// TwinCAT 3 PLC project CutomKeypadPLC
// ProgramVersion: 3.1.4023.0
// CompilerDefines: VISU_USEWSTRING
// libraries:
//   Tc2_Standard, * (Beckhoff Automation GmbH)
//   Tc2_System, * (Beckhoff Automation GmbH)
//   Tc3_Module, * (Beckhoff Automation GmbH)
//   VisuDialogs, * (System)
//   VisuSymbols,3.5.10.0,System
// project tree:
//   / GlobalTextList.TcGTLO, PlcTask.TcTTO, Visualization Manager.TcVMO (not stored), VISU_TASK.TcTTO
//   POUs/ MAIN.TcPOU
//   VISUs/ Custom_Keypad.TcVIS, Custom_Numpad.TcVIS, Visualization.TcVIS
// real-time tasks:
//   TASK PlcTask: cycle T#10ms, priority 20, ADS port 350
//   TASK VISU_TASK: cycle T#200000us, priority 30, ADS port 351

CONFIGURATION CutomKeypadPLC
    RESOURCE PLC ON TwinCAT3
        TASK PlcTask(INTERVAL := T#10ms, PRIORITY := 20);
        TASK VISU_TASK(INTERVAL := T#200000us, PRIORITY := 30);
        PROGRAM MAIN WITH PlcTask : MAIN;
        PROGRAM VisuElems_Visu_Prg WITH VISU_TASK : VisuElems.Visu_Prg;
    END_RESOURCE
END_CONFIGURATION

// ---- POUs/MAIN.TcPOU
(*	| author		| Beckhoff Automation Poland	|	*)
(* 	-------------------------------------------------	*)
(*	| wersion		| 1.0							|	*)
(* 	-------------------------------------------------	*)
(*	| TC version	| 3.1.4024.7					| 	*)
(* 	-------------------------------------------------	*)
(*	| date			| 19.05.2020					|	*)
(* 	-------------------------------------------------	*)
(*	| description	| custom keypad with hotkeys	|  	*)

PROGRAM MAIN
VAR
	iTest 	: INT;
	sTest	: STRING;
END_VAR

END_PROGRAM

// ---- GlobalTextList.TcGTLO
TEXTLIST GlobalTextList
  338 = '!'
  340 = '"'
  991 = '#'
  344 = '$'
  346 = '%'
  189 = '%s'
  169 = '&'
  992 = "'"
  174 = '('
  177 = ')'
  333 = '*'
  332 = '+'
  90 = '+/-'
  153 = ','
  157 = '-'
  155 = '.'
  171 = '/'
  179 = '0'
  337 = '1'
  339 = '2'
  341 = '3'
  343 = '4'
  345 = '5'
  347 = '6'
  170 = '7'
  172 = '8'
  176 = '9'
  156 = ':'
  154 = ';'
  137 = '<'
  181 = '='
  138 = '>'
  184 = '?'
  993 = '@'
  160 = 'a'
  161 = 'A'
  147 = 'b'
  148 = 'B'
  781 = 'Back'
  92 = 'Backspace'
  143 = 'c'
  144 = 'C'
  780 = 'Clear'
  164 = 'd'
  974 = 'D'
  998 = 'e'
  999 = 'E'
  253 = 'Enter number: %i'
  452 = 'Enter text: %s'
  779 = 'ESC'
  975 = 'f'
  976 = 'F'
  977 = 'g'
  978 = 'G'
  979 = 'h'
  980 = 'H'
  1008 = 'i'
  1009 = 'I'
  981 = 'j'
  982 = 'J'
  983 = 'k'
  984 = 'K'
  985 = 'l'
  986 = 'L'
  151 = 'm'
  152 = 'M'
  192 = 'Max:'
  191 = 'Min:'
  149 = 'n'
  150 = 'N'
  1010 = 'o'
  1011 = 'O'
  778 = 'OK'
  1012 = 'p'
  1013 = 'P'
  994 = 'q'
  995 = 'Q'
  1000 = 'r'
  1001 = 'R'
  162 = 's'
  163 = 'S'
  782 = 'Shift'
  783 = 'Space'
  1002 = 't'
  1003 = 'T'
  1006 = 'u'
  1007 = 'U'
  145 = 'v'
  146 = 'V'
  996 = 'w'
  997 = 'W'
  141 = 'x'
  142 = 'X'
  139 = 'y'
  140 = 'Y'
  1004 = 'z'
  1005 = 'Z'
  787 = '['
  187 = '\\'
  788 = ']'
  335 = '^'
  158 = '_'
  786 = '{'
  790 = '|'
  789 = '}'
  334 = '~'
  108 = '§'
  84 = '°'
  19 = '²'
  23 = '³'
  186 = '´'
  35 = 'ä'
  81 = 'Ä'
  29 = 'ö'
  34 = 'Ö'
  82 = 'ü'
  83 = 'Ü'
  109 = 'ß'
  28 = '€'
END_TEXTLIST

// ---- VISUs/Custom_Keypad.TcVIS
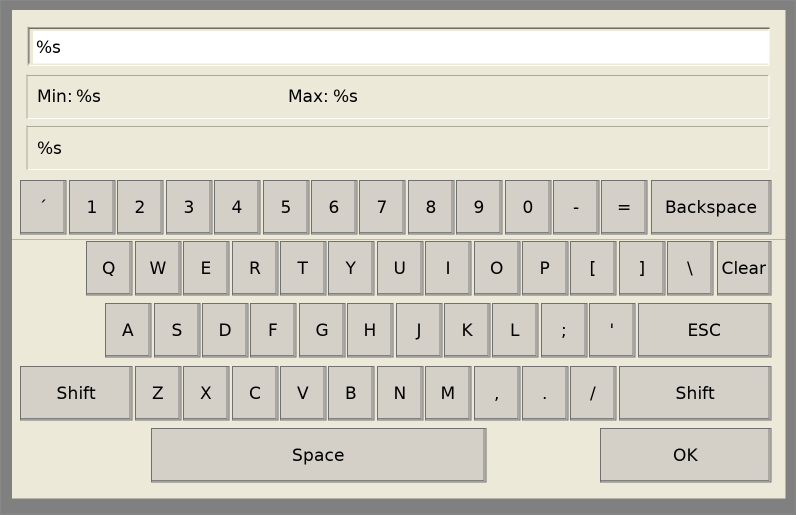
VISUALIZATION Custom_Keypad  // 796x515
VAR_INPUT
	stVariableValue : STRING;
	stMin : STRING;
	stMax : STRING;
	stTitle : STRING;
	flags : DWORD;
END_VAR
VAR
	bInit : BOOL;
	bShift : BOOL;
	stMessage : STRING;
	stOutputValue : STRING;
END_VAR
    Rectangle (0,0 796x515)
    Rectangle (12,169 773x70)
    Rectangle (12,240 773x62)
    Rectangle (12,301 773x63)
    Rectangle (12,364 773x62)
    Rectangle (12,423 773x75)
    Button (600,428 171x54), "OK"
        OnMouseDown: CloseDialog Dialog=Custom_Keypad, Result=OK, NumpadKeypad=True, NumpadKeypadSet=True
    Button (638,303 133x54), "ESC"
        OnMouseDown: CloseDialog Dialog=Custom_Keypad, Result=Cancel, NumpadKeypad=True, NumpadKeypadSet=True
    Button (717,241 54x54), "Clear"
        OnMouseDown: execute { stVariableValue := ''; stOutputValue := ''; }
    Button (651,180 120x54), "Backspace"
        OnMouseDown: execute { VisuDlg_CheckedBack(stOutputValue, stVariableValue, bInit); }
    Button (619,366 152x54), "Shift"
        OnMouseDown: toggle bShift
    Button (151,428 335x54), "Space"
        OnMouseDown: execute { VisuDlg_CheckedAppend(stOutputValue, stVariableValue, bInit, (flags AND VisuElems.Visu_InputFlags.Password) = 1, ' '); }
    Button (667,241 46x54), "|", invisible if: NOT bShift
        OnMouseDown: execute { VisuDlg_CheckedAppend(stOutputValue, stVariableValue, bInit, (flags AND VisuElems.Visu_InputFlags.Password) = 1, '|'); }
    Button (474,366 46x54), "<", invisible if: NOT bShift
        OnMouseDown: execute { VisuDlg_CheckedAppend(stOutputValue, stVariableValue, bInit, (flags AND VisuElems.Visu_InputFlags.Password) = 1, '<'); }
    Button (522,366 46x54), ">", invisible if: NOT bShift
        OnMouseDown: execute { VisuDlg_CheckedAppend(stOutputValue, stVariableValue, bInit, (flags AND VisuElems.Visu_InputFlags.Password) = 1, '>'); }
    Button (328,241 46x54), "y", invisible if: NOT bShift
        OnMouseDown: execute { VisuDlg_CheckedAppend(stOutputValue, stVariableValue, bInit, (flags AND VisuElems.Visu_InputFlags.Password) = 1, 'y'); }
    Button (328,241 46x54), "Y", invisible if: bShift
        OnMouseDown: execute { VisuDlg_CheckedAppend(stOutputValue, stVariableValue, bInit, (flags AND VisuElems.Visu_InputFlags.Password) = 1, 'Y'); }
    Button (183,366 46x54), "x", invisible if: NOT bShift
        OnMouseDown: execute { VisuDlg_CheckedAppend(stOutputValue, stVariableValue, bInit, (flags AND VisuElems.Visu_InputFlags.Password) = 1, 'x'); }
    Button (183,366 46x54), "X", invisible if: bShift
        OnMouseDown: execute { VisuDlg_CheckedAppend(stOutputValue, stVariableValue, bInit, (flags AND VisuElems.Visu_InputFlags.Password) = 1, 'X'); }
    Button (232,366 46x54), "c", invisible if: NOT bShift
        OnMouseDown: execute { VisuDlg_CheckedAppend(stOutputValue, stVariableValue, bInit, (flags AND VisuElems.Visu_InputFlags.Password) = 1, 'c'); }
    Button (232,366 46x54), "C", invisible if: bShift
        OnMouseDown: execute { VisuDlg_CheckedAppend(stOutputValue, stVariableValue, bInit, (flags AND VisuElems.Visu_InputFlags.Password) = 1, 'C'); }
    Button (280,366 46x54), "v", invisible if: NOT bShift
        OnMouseDown: execute { VisuDlg_CheckedAppend(stOutputValue, stVariableValue, bInit, (flags AND VisuElems.Visu_InputFlags.Password) = 1, 'v'); }
    Button (280,366 46x54), "V", invisible if: bShift
        OnMouseDown: execute { VisuDlg_CheckedAppend(stOutputValue, stVariableValue, bInit, (flags AND VisuElems.Visu_InputFlags.Password) = 1, 'V'); }
    Button (328,366 46x54), "b", invisible if: NOT bShift
        OnMouseDown: execute { VisuDlg_CheckedAppend(stOutputValue, stVariableValue, bInit, (flags AND VisuElems.Visu_InputFlags.Password) = 1, 'b'); }
    Button (328,366 46x54), "B", invisible if: bShift
        OnMouseDown: execute { VisuDlg_CheckedAppend(stOutputValue, stVariableValue, bInit, (flags AND VisuElems.Visu_InputFlags.Password) = 1, 'B'); }
    Button (377,366 46x54), "n", invisible if: NOT bShift
        OnMouseDown: execute { VisuDlg_CheckedAppend(stOutputValue, stVariableValue, bInit, (flags AND VisuElems.Visu_InputFlags.Password) = 1, 'n'); }
    Button (377,366 46x54), "N", invisible if: bShift
        OnMouseDown: execute { VisuDlg_CheckedAppend(stOutputValue, stVariableValue, bInit, (flags AND VisuElems.Visu_InputFlags.Password) = 1, 'N'); }
    Button (425,366 46x54), "m", invisible if: NOT bShift
        OnMouseDown: execute { VisuDlg_CheckedAppend(stOutputValue, stVariableValue, bInit, (flags AND VisuElems.Visu_InputFlags.Password) = 1, 'm'); }
    Button (425,366 46x54), "M", invisible if: bShift
        OnMouseDown: execute { VisuDlg_CheckedAppend(stOutputValue, stVariableValue, bInit, (flags AND VisuElems.Visu_InputFlags.Password) = 1, 'M'); }
    Button (541,303 46x54), ":", invisible if: NOT bShift
        OnMouseDown: execute { VisuDlg_CheckedAppend(stOutputValue, stVariableValue, bInit, (flags AND VisuElems.Visu_InputFlags.Password) = 1, ':'); }
    Button (553,180 46x54), "_", invisible if: NOT bShift
        OnMouseDown: execute { VisuDlg_CheckedAppend(stOutputValue, stVariableValue, bInit, (flags AND VisuElems.Visu_InputFlags.Password) = 1, '_'); }
    Button (105,303 46x54), "a", invisible if: NOT bShift
        OnMouseDown: execute { VisuDlg_CheckedAppend(stOutputValue, stVariableValue, bInit, (flags AND VisuElems.Visu_InputFlags.Password) = 1, 'a'); }
    Button (105,303 46x54), "A", invisible if: bShift
        OnMouseDown: execute { VisuDlg_CheckedAppend(stOutputValue, stVariableValue, bInit, (flags AND VisuElems.Visu_InputFlags.Password) = 1, 'A'); }
    Button (154,303 46x54), "s", invisible if: NOT bShift
        OnMouseDown: execute { VisuDlg_CheckedAppend(stOutputValue, stVariableValue, bInit, (flags AND VisuElems.Visu_InputFlags.Password) = 1, 's'); }
    Button (154,303 46x54), "S", invisible if: bShift
        OnMouseDown: execute { VisuDlg_CheckedAppend(stOutputValue, stVariableValue, bInit, (flags AND VisuElems.Visu_InputFlags.Password) = 1, 'S'); }
    Button (202,303 46x54), "d", invisible if: NOT bShift
        OnMouseDown: execute { VisuDlg_CheckedAppend(stOutputValue, stVariableValue, bInit, (flags AND VisuElems.Visu_InputFlags.Password) = 1, 'd'); }
    Button (202,303 46x54), "D", invisible if: bShift
        OnMouseDown: execute { VisuDlg_CheckedAppend(stOutputValue, stVariableValue, bInit, (flags AND VisuElems.Visu_InputFlags.Password) = 1, 'D'); }
    Button (250,303 46x54), "f", invisible if: NOT bShift
        OnMouseDown: execute { VisuDlg_CheckedAppend(stOutputValue, stVariableValue, bInit, (flags AND VisuElems.Visu_InputFlags.Password) = 1, 'f'); }
    Button (250,303 46x54), "F", invisible if: bShift
        OnMouseDown: execute { VisuDlg_CheckedAppend(stOutputValue, stVariableValue, bInit, (flags AND VisuElems.Visu_InputFlags.Password) = 1, 'F'); }
    Button (299,303 46x54), "g", invisible if: NOT bShift
        OnMouseDown: execute { VisuDlg_CheckedAppend(stOutputValue, stVariableValue, bInit, (flags AND VisuElems.Visu_InputFlags.Password) = 1, 'g'); }
    Button (299,303 46x54), "G", invisible if: bShift
        OnMouseDown: execute { VisuDlg_CheckedAppend(stOutputValue, stVariableValue, bInit, (flags AND VisuElems.Visu_InputFlags.Password) = 1, 'G'); }
    Button (347,303 46x54), "h", invisible if: NOT bShift
        OnMouseDown: execute { VisuDlg_CheckedAppend(stOutputValue, stVariableValue, bInit, (flags AND VisuElems.Visu_InputFlags.Password) = 1, 'h'); }
    Button (347,303 46x54), "H", invisible if: bShift
        OnMouseDown: execute { VisuDlg_CheckedAppend(stOutputValue, stVariableValue, bInit, (flags AND VisuElems.Visu_InputFlags.Password) = 1, 'H'); }
    Button (396,303 46x54), "j", invisible if: NOT bShift
        OnMouseDown: execute { VisuDlg_CheckedAppend(stOutputValue, stVariableValue, bInit, (flags AND VisuElems.Visu_InputFlags.Password) = 1, 'j'); }
    Button (396,303 46x54), "J", invisible if: bShift
        OnMouseDown: execute { VisuDlg_CheckedAppend(stOutputValue, stVariableValue, bInit, (flags AND VisuElems.Visu_InputFlags.Password) = 1, 'J'); }
    Button (444,303 46x54), "k", invisible if: NOT bShift
        OnMouseDown: execute { VisuDlg_CheckedAppend(stOutputValue, stVariableValue, bInit, (flags AND VisuElems.Visu_InputFlags.Password) = 1, 'k'); }
    Button (444,303 46x54), "K", invisible if: bShift
        OnMouseDown: execute { VisuDlg_CheckedAppend(stOutputValue, stVariableValue, bInit, (flags AND VisuElems.Visu_InputFlags.Password) = 1, 'K'); }
    Button (492,303 46x54), "l", invisible if: NOT bShift
        OnMouseDown: execute { VisuDlg_CheckedAppend(stOutputValue, stVariableValue, bInit, (flags AND VisuElems.Visu_InputFlags.Password) = 1, 'l'); }
    Button (492,303 46x54), "L", invisible if: bShift
        OnMouseDown: execute { VisuDlg_CheckedAppend(stOutputValue, stVariableValue, bInit, (flags AND VisuElems.Visu_InputFlags.Password) = 1, 'L'); }
    Button (166,180 46x54), "#", invisible if: NOT bShift
        OnMouseDown: execute { VisuDlg_CheckedAppend(stOutputValue, stVariableValue, bInit, (flags AND VisuElems.Visu_InputFlags.Password) = 1, '#'); }
    Button (117,180 46x54), "@", invisible if: NOT bShift
        OnMouseDown: execute { VisuDlg_CheckedAppend(stOutputValue, stVariableValue, bInit, (flags AND VisuElems.Visu_InputFlags.Password) = 1, '@'); }
    Button (86,241 46x54), "q", invisible if: NOT bShift
        OnMouseDown: execute { VisuDlg_CheckedAppend(stOutputValue, stVariableValue, bInit, (flags AND VisuElems.Visu_InputFlags.Password) = 1, 'q'); }
    Button (86,241 46x54), "Q", invisible if: bShift
        OnMouseDown: execute { VisuDlg_CheckedAppend(stOutputValue, stVariableValue, bInit, (flags AND VisuElems.Visu_InputFlags.Password) = 1, 'Q'); }
    Button (135,241 46x54), "w", invisible if: NOT bShift
        OnMouseDown: execute { VisuDlg_CheckedAppend(stOutputValue, stVariableValue, bInit, (flags AND VisuElems.Visu_InputFlags.Password) = 1, 'w'); }
    Button (135,241 46x54), "W", invisible if: bShift
        OnMouseDown: execute { VisuDlg_CheckedAppend(stOutputValue, stVariableValue, bInit, (flags AND VisuElems.Visu_InputFlags.Password) = 1, 'W'); }
    Button (183,241 46x54), "e", invisible if: NOT bShift
        OnMouseDown: execute { VisuDlg_CheckedAppend(stOutputValue, stVariableValue, bInit, (flags AND VisuElems.Visu_InputFlags.Password) = 1, 'e'); }
    Button (183,241 46x54), "E", invisible if: bShift
        OnMouseDown: execute { VisuDlg_CheckedAppend(stOutputValue, stVariableValue, bInit, (flags AND VisuElems.Visu_InputFlags.Password) = 1, 'E'); }
    Button (232,241 46x54), "r", invisible if: NOT bShift
        OnMouseDown: execute { VisuDlg_CheckedAppend(stOutputValue, stVariableValue, bInit, (flags AND VisuElems.Visu_InputFlags.Password) = 1, 'r'); }
    Button (232,241 46x54), "R", invisible if: bShift
        OnMouseDown: execute { VisuDlg_CheckedAppend(stOutputValue, stVariableValue, bInit, (flags AND VisuElems.Visu_InputFlags.Password) = 1, 'R'); }
    Button (280,241 46x54), "t", invisible if: NOT bShift
        OnMouseDown: execute { VisuDlg_CheckedAppend(stOutputValue, stVariableValue, bInit, (flags AND VisuElems.Visu_InputFlags.Password) = 1, 't'); }
    Button (280,241 46x54), "T", invisible if: bShift
        OnMouseDown: execute { VisuDlg_CheckedAppend(stOutputValue, stVariableValue, bInit, (flags AND VisuElems.Visu_InputFlags.Password) = 1, 'T'); }
    Button (135,366 46x54), "z", invisible if: NOT bShift
        OnMouseDown: execute { VisuDlg_CheckedAppend(stOutputValue, stVariableValue, bInit, (flags AND VisuElems.Visu_InputFlags.Password) = 1, 'z'); }
    Button (135,366 46x54), "Z", invisible if: bShift
        OnMouseDown: execute { VisuDlg_CheckedAppend(stOutputValue, stVariableValue, bInit, (flags AND VisuElems.Visu_InputFlags.Password) = 1, 'Z'); }
    Button (377,241 46x54), "u", invisible if: NOT bShift
        OnMouseDown: execute { VisuDlg_CheckedAppend(stOutputValue, stVariableValue, bInit, (flags AND VisuElems.Visu_InputFlags.Password) = 1, 'u'); }
    Button (377,241 46x54), "U", invisible if: bShift
        OnMouseDown: execute { VisuDlg_CheckedAppend(stOutputValue, stVariableValue, bInit, (flags AND VisuElems.Visu_InputFlags.Password) = 1, 'U'); }
    Button (425,241 46x54), "i", invisible if: NOT bShift
        OnMouseDown: execute { VisuDlg_CheckedAppend(stOutputValue, stVariableValue, bInit, (flags AND VisuElems.Visu_InputFlags.Password) = 1, 'i'); }
    Button (425,241 46x54), "I", invisible if: bShift
        OnMouseDown: execute { VisuDlg_CheckedAppend(stOutputValue, stVariableValue, bInit, (flags AND VisuElems.Visu_InputFlags.Password) = 1, 'I'); }
    Button (474,241 46x54), "o", invisible if: NOT bShift
        OnMouseDown: execute { VisuDlg_CheckedAppend(stOutputValue, stVariableValue, bInit, (flags AND VisuElems.Visu_InputFlags.Password) = 1, 'o'); }
    Button (474,241 46x54), "O", invisible if: bShift
        OnMouseDown: execute { VisuDlg_CheckedAppend(stOutputValue, stVariableValue, bInit, (flags AND VisuElems.Visu_InputFlags.Password) = 1, 'O'); }
    Button (522,241 46x54), "p", invisible if: NOT bShift
        OnMouseDown: execute { VisuDlg_CheckedAppend(stOutputValue, stVariableValue, bInit, (flags AND VisuElems.Visu_InputFlags.Password) = 1, 'p'); }
    Button (522,241 46x54), "P", invisible if: bShift
        OnMouseDown: execute { VisuDlg_CheckedAppend(stOutputValue, stVariableValue, bInit, (flags AND VisuElems.Visu_InputFlags.Password) = 1, 'P'); }
    Button (601,180 46x54), "+", invisible if: NOT bShift
        OnMouseDown: execute { VisuDlg_CheckedAppend(stOutputValue, stVariableValue, bInit, (flags AND VisuElems.Visu_InputFlags.Password) = 1, '+'); }
    Button (408,180 46x54), "*", invisible if: NOT bShift
        OnMouseDown: execute { VisuDlg_CheckedAppend(stOutputValue, stVariableValue, bInit, (flags AND VisuElems.Visu_InputFlags.Password) = 1, '*'); }
    Button (20,180 46x54), "~", invisible if: NOT bShift
        OnMouseDown: execute { VisuDlg_CheckedAppend(stOutputValue, stVariableValue, bInit, (flags AND VisuElems.Visu_InputFlags.Password) = 1, '~'); }
    Button (311,180 46x54), "^", invisible if: NOT bShift
        OnMouseDown: execute { VisuDlg_CheckedAppend(stOutputValue, stVariableValue, bInit, (flags AND VisuElems.Visu_InputFlags.Password) = 1, '^'); }
    Button (69,180 46x54), "!", invisible if: NOT bShift
        OnMouseDown: execute { VisuDlg_CheckedAppend(stOutputValue, stVariableValue, bInit, (flags AND VisuElems.Visu_InputFlags.Password) = 1, '!'); }
    Button (589,303 46x54), """, invisible if: NOT bShift
        OnMouseDown: execute { VisuDlg_CheckedAppend(stOutputValue, stVariableValue, bInit, (flags AND VisuElems.Visu_InputFlags.Password) = 1, '"'); }
    Button (214,180 46x54), "$", invisible if: NOT bShift
        OnMouseDown: execute { VisuDlg_CheckedAppend(stOutputValue, stVariableValue, bInit, (flags AND VisuElems.Visu_InputFlags.Password) = 1, '$$'); }
    Button (263,180 46x54), "%", invisible if: NOT bShift
        OnMouseDown: execute { VisuDlg_CheckedAppend(stOutputValue, stVariableValue, bInit, (flags AND VisuElems.Visu_InputFlags.Password) = 1, '%'); }
    Button (359,180 46x54), "&", invisible if: NOT bShift
        OnMouseDown: execute { VisuDlg_CheckedAppend(stOutputValue, stVariableValue, bInit, (flags AND VisuElems.Visu_InputFlags.Password) = 1, '&'); }
    Button (456,180 46x54), "(", invisible if: NOT bShift
        OnMouseDown: execute { VisuDlg_CheckedAppend(stOutputValue, stVariableValue, bInit, (flags AND VisuElems.Visu_InputFlags.Password) = 1, '('); }
    Button (505,180 46x54), ")", invisible if: NOT bShift
        OnMouseDown: execute { VisuDlg_CheckedAppend(stOutputValue, stVariableValue, bInit, (flags AND VisuElems.Visu_InputFlags.Password) = 1, ')'); }
    Button (570,366 46x54), "?", invisible if: NOT bShift
        OnMouseDown: execute { VisuDlg_CheckedAppend(stOutputValue, stVariableValue, bInit, (flags AND VisuElems.Visu_InputFlags.Password) = 1, '?'); }
    Rectangle (12,72 773x97)
    Rectangle (34,132 734x32), "%s", text variable: stMessage
    Rectangle (12,10 773x62)
    Polyline (27,169) (27,126) (769,126)
    Polyline (27,118) (27,75) (769,75)
    Polyline (28,65) (28,27) (769,27)
    Polyline (28,169) (769,169) (769,126)
    Polyline (28,118) (769,118) (769,75)
    Polyline (29,65) (769,65) (769,28)
    Polyline (29,63) (29,28) (769,28)
    Rectangle (33,31 736x32), "%s", text variable: stOutputValue
    Rectangle (34,80 42x32), "Min:", text variable: stMin, invisible if: LEN(stMin) = 0
    Rectangle (73,80 157x32), "%s", text variable: stMin, invisible if: LEN(stMin) = 0
    Rectangle (285,80 45x32), "Max:", text variable: stMin, invisible if: LEN(stMax) = 0
    Rectangle (330,80 217x32), "%s", text variable: stMax, invisible if: LEN(stMax) = 0
    Button (20,180 46x54), "´", invisible if: bShift
        OnMouseDown: execute { VisuDlg_CheckedAppend(stOutputValue, stVariableValue, bInit, (flags AND VisuElems.Visu_InputFlags.Password) = 1, '´'); }
    Button (69,180 46x54), "1", invisible if: bShift
        OnMouseDown: execute { VisuDlg_CheckedAppend(stOutputValue, stVariableValue, bInit, (flags AND VisuElems.Visu_InputFlags.Password) = 1, '1'); }
    Button (117,180 46x54), "2", invisible if: bShift
        OnMouseDown: execute { VisuDlg_CheckedAppend(stOutputValue, stVariableValue, bInit, (flags AND VisuElems.Visu_InputFlags.Password) = 1, '2'); }
    Button (166,180 46x54), "3", invisible if: bShift
        OnMouseDown: execute { VisuDlg_CheckedAppend(stOutputValue, stVariableValue, bInit, (flags AND VisuElems.Visu_InputFlags.Password) = 1, '3'); }
    Button (214,180 46x54), "4", invisible if: bShift
        OnMouseDown: execute { VisuDlg_CheckedAppend(stOutputValue, stVariableValue, bInit, (flags AND VisuElems.Visu_InputFlags.Password) = 1, '4'); }
    Button (263,180 46x54), "5", invisible if: bShift
        OnMouseDown: execute { VisuDlg_CheckedAppend(stOutputValue, stVariableValue, bInit, (flags AND VisuElems.Visu_InputFlags.Password) = 1, '5'); }
    Button (311,180 46x54), "6", invisible if: bShift
        OnMouseDown: execute { VisuDlg_CheckedAppend(stOutputValue, stVariableValue, bInit, (flags AND VisuElems.Visu_InputFlags.Password) = 1, '6'); }
    Button (359,180 46x54), "7", invisible if: bShift
        OnMouseDown: execute { VisuDlg_CheckedAppend(stOutputValue, stVariableValue, bInit, (flags AND VisuElems.Visu_InputFlags.Password) = 1, '7'); }
    Button (408,180 46x54), "8", invisible if: bShift
        OnMouseDown: execute { VisuDlg_CheckedAppend(stOutputValue, stVariableValue, bInit, (flags AND VisuElems.Visu_InputFlags.Password) = 1, '8'); }
    Button (456,180 46x54), "9", invisible if: bShift
        OnMouseDown: execute { VisuDlg_CheckedAppend(stOutputValue, stVariableValue, bInit, (flags AND VisuElems.Visu_InputFlags.Password) = 1, '9'); }
    Button (505,180 46x54), "0", invisible if: bShift
        OnMouseDown: execute { VisuDlg_CheckedAppend(stOutputValue, stVariableValue, bInit, (flags AND VisuElems.Visu_InputFlags.Password) = 1, '0'); }
    Button (553,180 46x54), "-", invisible if: bShift
        OnMouseDown: execute { VisuDlg_CheckedAppend(stOutputValue, stVariableValue, bInit, (flags AND VisuElems.Visu_InputFlags.Password) = 1, '-'); }
    Button (601,180 46x54), "=", invisible if: bShift
        OnMouseDown: execute { VisuDlg_CheckedAppend(stOutputValue, stVariableValue, bInit, (flags AND VisuElems.Visu_InputFlags.Password) = 1, '='); }
    Button (570,241 46x54), "{", invisible if: NOT bShift
        OnMouseDown: execute { VisuDlg_CheckedAppend(stOutputValue, stVariableValue, bInit, (flags AND VisuElems.Visu_InputFlags.Password) = 1, '{'); }
    Button (570,241 46x54), "[", invisible if: bShift
        OnMouseDown: execute { VisuDlg_CheckedAppend(stOutputValue, stVariableValue, bInit, (flags AND VisuElems.Visu_InputFlags.Password) = 1, '['); }
    Button (619,241 46x54), "}", invisible if: NOT bShift
        OnMouseDown: execute { VisuDlg_CheckedAppend(stOutputValue, stVariableValue, bInit, (flags AND VisuElems.Visu_InputFlags.Password) = 1, '}'); }
    Button (619,241 46x54), "]", invisible if: bShift
        OnMouseDown: execute { VisuDlg_CheckedAppend(stOutputValue, stVariableValue, bInit, (flags AND VisuElems.Visu_InputFlags.Password) = 1, ']'); }
    Button (667,241 46x54), "\", invisible if: bShift
        OnMouseDown: execute { VisuDlg_CheckedAppend(stOutputValue, stVariableValue, bInit, (flags AND VisuElems.Visu_InputFlags.Password) = 1, '\'); }
    Button (541,303 46x54), ";", invisible if: bShift
        OnMouseDown: execute { VisuDlg_CheckedAppend(stOutputValue, stVariableValue, bInit, (flags AND VisuElems.Visu_InputFlags.Password) = 1, ';'); }
    Button (589,303 46x54), "'", invisible if: bShift
        OnMouseDown: execute { VisuDlg_CheckedAppend(stOutputValue, stVariableValue, bInit, (flags AND VisuElems.Visu_InputFlags.Password) = 1, '$''); }
    Button (474,366 46x54), ",", invisible if: bShift
        OnMouseDown: execute { VisuDlg_CheckedAppend(stOutputValue, stVariableValue, bInit, (flags AND VisuElems.Visu_InputFlags.Password) = 1, ','); }
    Button (522,366 46x54), ".", invisible if: bShift
        OnMouseDown: execute { VisuDlg_CheckedAppend(stOutputValue, stVariableValue, bInit, (flags AND VisuElems.Visu_InputFlags.Password) = 1, '.'); }
    Button (570,366 46x54), "/", invisible if: bShift
        OnMouseDown: execute { VisuDlg_CheckedAppend(stOutputValue, stVariableValue, bInit, (flags AND VisuElems.Visu_InputFlags.Password) = 1, '/'); }
    Button (20,366 112x54), "Shift"
        OnMouseDown: toggle bShift
    hotkey HotkeyInput Id=481083523072, Key=KeyDown=True, KeyName=BACKSPACE, ActionToExecute=Action=STSnippet=VisuDlg_CheckedBack(stOutputValue, stVariableValue, bInit);, VisuElemId=-1
    hotkey HotkeyInput Id=481084571648, Key=KeyDown=True, KeyName=DELETE, ActionToExecute=Action=STSnippet=stVariableValue := ''; stOutputValue := '';, VisuElemId=-1
    hotkey HotkeyInput Id=481085620224, Key=KeyDown=True, KeyName=ESCAPE, ActionToExecute=Action=Dialog=Custom_Keypad, Result=Cancel, NumpadKeypad=True, NumpadKeypadSet=True, VisuElemId=-1
    hotkey HotkeyInput Id=481086668800, Key=KeyDown=True, KeyName=SPACE, ActionToExecute=Action=STSnippet=VisuDlg_CheckedAppend(stOutputValue, stVariableValue, bInit, (flags AND VisuElems.Visu_InputFlags.Password) = 1, ' ');, VisuElemId=-1
    hotkey HotkeyInput Id=481087717376, Key=Modifiers=1, KeyDown=True, KeyName=SPACE, ActionToExecute=Action=ToggleVariable=bShift, VisuElemId=-1
    hotkey HotkeyInput Id=481088765952, Key=KeyDown=True, KeyName=RETURN_KEY, ActionToExecute=Action=Dialog=Custom_Keypad, Result=OK, NumpadKeypad=True, NumpadKeypadSet=True, VisuElemId=-1
    hotkey HotkeyInput Id=481089814528, Key=KeyDown=True, KeyName=1, ActionToExecute=Action=STSnippet=IF bShift THEN VisuDlg_CheckedAppend(stOutputValue, stVariableValue, bInit, (flags AND VisuElems.Visu_InputFlags.Password) = 1, '!'); ELSE VisuDlg_CheckedAppend(stOutputValue, stVariableValue, bInit, (flags AND VisuElems.Visu_InputFlags.Password) = 1, '1'); END_IF, VisuElemId=-1
    hotkey HotkeyInput Id=481090863104, Key=KeyDown=True, KeyName=2, ActionToExecute=Action=STSnippet=IF bShift THEN VisuDlg_CheckedAppend(stOutputValue, stVariableValue, bInit, (flags AND VisuElems.Visu_InputFlags.Password) = 1, '@'); ELSE VisuDlg_CheckedAppend(stOutputValue, stVariableValue, bInit, (flags AND VisuElems.Visu_InputFlags.Password) = 1, '2'); END_IF, VisuElemId=-1
    hotkey HotkeyInput Id=481091911680, Key=KeyDown=True, KeyName=3, ActionToExecute=Action=STSnippet=IF bShift THEN VisuDlg_CheckedAppend(stOutputValue, stVariableValue, bInit, (flags AND VisuElems.Visu_InputFlags.Password) = 1, '#'); ELSE VisuDlg_CheckedAppend(stOutputValue, stVariableValue, bInit, (flags AND VisuElems.Visu_InputFlags.Password) = 1, '3'); END_IF, VisuElemId=-1
    hotkey HotkeyInput Id=481092960256, Key=KeyDown=True, KeyName=4, ActionToExecute=Action=STSnippet=IF bShift THEN VisuDlg_CheckedAppend(stOutputValue, stVariableValue, bInit, (flags AND VisuElems.Visu_InputFlags.Password) = 1, '$$'); ELSE VisuDlg_CheckedAppend(stOutputValue, stVariableValue, bInit, (flags AND VisuElems.Visu_InputFlags.Password) = 1, '4'); END_IF, VisuElemId=-1
    hotkey HotkeyInput Id=481094008832, Key=KeyDown=True, KeyName=5, ActionToExecute=Action=STSnippet=IF bShift THEN VisuDlg_CheckedAppend(stOutputValue, stVariableValue, bInit, (flags AND VisuElems.Visu_InputFlags.Password) = 1, '%'); ELSE VisuDlg_CheckedAppend(stOutputValue, stVariableValue, bInit, (flags AND VisuElems.Visu_InputFlags.Password) = 1, '5'); END_IF, VisuElemId=-1
    hotkey HotkeyInput Id=481095057408, Key=KeyDown=True, KeyName=6, ActionToExecute=Action=STSnippet=IF bShift THEN VisuDlg_CheckedAppend(stOutputValue, stVariableValue, bInit, (flags AND VisuElems.Visu_InputFlags.Password) = 1, '^'); ELSE VisuDlg_CheckedAppend(stOutputValue, stVariableValue, bInit, (flags AND VisuElems.Visu_InputFlags.Password) = 1, '6'); END_IF, VisuElemId=-1
    hotkey HotkeyInput Id=481096105984, Key=KeyDown=True, KeyName=7, ActionToExecute=Action=STSnippet=IF bShift THEN VisuDlg_CheckedAppend(stOutputValue, stVariableValue, bInit, (flags AND VisuElems.Visu_InputFlags.Password) = 1, '&'); ELSE VisuDlg_CheckedAppend(stOutputValue, stVariableValue, bInit, (flags AND VisuElems.Visu_InputFlags.Password) = 1, '7'); END_IF, VisuElemId=-1
    hotkey HotkeyInput Id=481097154560, Key=KeyDown=True, KeyName=8, ActionToExecute=Action=STSnippet=IF bShift THEN VisuDlg_CheckedAppend(stOutputValue, stVariableValue, bInit, (flags AND VisuElems.Visu_InputFlags.Password) = 1, '*'); ELSE VisuDlg_CheckedAppend(stOutputValue, stVariableValue, bInit, (flags AND VisuElems.Visu_InputFlags.Password) = 1, '8'); END_IF, VisuElemId=-1
    hotkey HotkeyInput Id=481098203136, Key=KeyDown=True, KeyName=9, ActionToExecute=Action=STSnippet=IF bShift THEN VisuDlg_CheckedAppend(stOutputValue, stVariableValue, bInit, (flags AND VisuElems.Visu_InputFlags.Password) = 1, '('); ELSE VisuDlg_CheckedAppend(stOutputValue, stVariableValue, bInit, (flags AND VisuElems.Visu_InputFlags.Password) = 1, '9'); END_IF, VisuElemId=-1
    hotkey HotkeyInput Id=481099251712, Key=KeyDown=True, KeyName=0, ActionToExecute=Action=STSnippet=IF bShift THEN VisuDlg_CheckedAppend(stOutputValue, stVariableValue, bInit, (flags AND VisuElems.Visu_InputFlags.Password) = 1, ')'); ELSE VisuDlg_CheckedAppend(stOutputValue, stVariableValue, bInit, (flags AND VisuElems.Visu_InputFlags.Password) = 1, '0'); END_IF, VisuElemId=-1
    hotkey HotkeyInput Id=481100300288, Key=KeyDown=True, KeyName=SUBTRACT, ActionToExecute=Action=STSnippet=IF bShift THEN VisuDlg_CheckedAppend(stOutputValue, stVariableValue, bInit, (flags AND VisuElems.Visu_InputFlags.Password) = 1, '_'); ELSE VisuDlg_CheckedAppend(stOutputValue, stVariableValue, bInit, (flags AND VisuElems.Visu_InputFlags.Password) = 1, '-'); END_IF, VisuElemId=-1
    hotkey HotkeyInput Id=481101348864, Key=KeyDown=True, KeyName=ADDITION, ActionToExecute=Action=STSnippet=IF bShift THEN VisuDlg_CheckedAppend(stOutputValue, stVariableValue, bInit, (flags AND VisuElems.Visu_InputFlags.Password) = 1, '='); ELSE VisuDlg_CheckedAppend(stOutputValue, stVariableValue, bInit, (flags AND VisuElems.Visu_InputFlags.Password) = 1, '+'); END_IF, VisuElemId=-1
    hotkey HotkeyInput Id=481102397440, Key=KeyDown=True, KeyName=Q, ActionToExecute=Action=STSnippet=IF bShift THEN VisuDlg_CheckedAppend(stOutputValue, stVariableValue, bInit, (flags AND VisuElems.Visu_InputFlags.Password) = 1, 'q'); ELSE VisuDlg_CheckedAppend(stOutputValue, stVariableValue, bInit, (flags AND VisuElems.Visu_InputFlags.Password) = 1, 'Q'); END_IF, VisuElemId=-1
    hotkey HotkeyInput Id=481103446016, Key=KeyDown=True, KeyName=W, ActionToExecute=Action=STSnippet=IF bShift THEN VisuDlg_CheckedAppend(stOutputValue, stVariableValue, bInit, (flags AND VisuElems.Visu_InputFlags.Password) = 1, 'w'); ELSE VisuDlg_CheckedAppend(stOutputValue, stVariableValue, bInit, (flags AND VisuElems.Visu_InputFlags.Password) = 1, 'W'); END_IF, VisuElemId=-1
    hotkey HotkeyInput Id=481104494592, Key=KeyDown=True, KeyName=E, ActionToExecute=Action=STSnippet=IF bShift THEN VisuDlg_CheckedAppend(stOutputValue, stVariableValue, bInit, (flags AND VisuElems.Visu_InputFlags.Password) = 1, 'e'); ELSE VisuDlg_CheckedAppend(stOutputValue, stVariableValue, bInit, (flags AND VisuElems.Visu_InputFlags.Password) = 1, 'E'); END_IF, VisuElemId=-1
    hotkey HotkeyInput Id=481105543168, Key=KeyDown=True, KeyName=R, ActionToExecute=Action=STSnippet=IF bShift THEN VisuDlg_CheckedAppend(stOutputValue, stVariableValue, bInit, (flags AND VisuElems.Visu_InputFlags.Password) = 1, 'r'); ELSE VisuDlg_CheckedAppend(stOutputValue, stVariableValue, bInit, (flags AND VisuElems.Visu_InputFlags.Password) = 1, 'R'); END_IF, VisuElemId=-1
    hotkey HotkeyInput Id=481106591744, Key=KeyDown=True, KeyName=T, ActionToExecute=Action=STSnippet=IF bShift THEN VisuDlg_CheckedAppend(stOutputValue, stVariableValue, bInit, (flags AND VisuElems.Visu_InputFlags.Password) = 1, 't'); ELSE VisuDlg_CheckedAppend(stOutputValue, stVariableValue, bInit, (flags AND VisuElems.Visu_InputFlags.Password) = 1, 'T'); END_IF, VisuElemId=-1
    hotkey HotkeyInput Id=481107640320, Key=KeyDown=True, KeyName=Y, ActionToExecute=Action=STSnippet=IF bShift THEN VisuDlg_CheckedAppend(stOutputValue, stVariableValue, bInit, (flags AND VisuElems.Visu_InputFlags.Password) = 1, 'y'); ELSE VisuDlg_CheckedAppend(stOutputValue, stVariableValue, bInit, (flags AND VisuElems.Visu_InputFlags.Password) = 1, 'Y'); END_IF, VisuElemId=-1
    hotkey HotkeyInput Id=481108688896, Key=KeyDown=True, KeyName=U, ActionToExecute=Action=STSnippet=IF bShift THEN VisuDlg_CheckedAppend(stOutputValue, stVariableValue, bInit, (flags AND VisuElems.Visu_InputFlags.Password) = 1, 'u'); ELSE VisuDlg_CheckedAppend(stOutputValue, stVariableValue, bInit, (flags AND VisuElems.Visu_InputFlags.Password) = 1, 'U'); END_IF, VisuElemId=-1
    hotkey HotkeyInput Id=481109737472, Key=KeyDown=True, KeyName=I, ActionToExecute=Action=STSnippet=IF bShift THEN VisuDlg_CheckedAppend(stOutputValue, stVariableValue, bInit, (flags AND VisuElems.Visu_InputFlags.Password) = 1, 'i'); ELSE VisuDlg_CheckedAppend(stOutputValue, stVariableValue, bInit, (flags AND VisuElems.Visu_InputFlags.Password) = 1, 'I'); END_IF, VisuElemId=-1
    hotkey HotkeyInput Id=481110786048, Key=KeyDown=True, KeyName=O, ActionToExecute=Action=STSnippet=IF bShift THEN VisuDlg_CheckedAppend(stOutputValue, stVariableValue, bInit, (flags AND VisuElems.Visu_InputFlags.Password) = 1, 'o'); ELSE VisuDlg_CheckedAppend(stOutputValue, stVariableValue, bInit, (flags AND VisuElems.Visu_InputFlags.Password) = 1, 'O'); END_IF, VisuElemId=-1
    hotkey HotkeyInput Id=481111834624, Key=KeyDown=True, KeyName=P, ActionToExecute=Action=STSnippet=IF bShift THEN VisuDlg_CheckedAppend(stOutputValue, stVariableValue, bInit, (flags AND VisuElems.Visu_InputFlags.Password) = 1, 'p'); ELSE VisuDlg_CheckedAppend(stOutputValue, stVariableValue, bInit, (flags AND VisuElems.Visu_InputFlags.Password) = 1, 'P'); END_IF, VisuElemId=-1
    hotkey HotkeyInput Id=481112883200, Key=KeyDown=True, KeyName=A, ActionToExecute=Action=STSnippet=IF bShift THEN VisuDlg_CheckedAppend(stOutputValue, stVariableValue, bInit, (flags AND VisuElems.Visu_InputFlags.Password) = 1, 'a'); ELSE VisuDlg_CheckedAppend(stOutputValue, stVariableValue, bInit, (flags AND VisuElems.Visu_InputFlags.Password) = 1, 'A'); END_IF, VisuElemId=-1
    hotkey HotkeyInput Id=481113931776, Key=KeyDown=True, KeyName=S, ActionToExecute=Action=STSnippet=IF bShift THEN VisuDlg_CheckedAppend(stOutputValue, stVariableValue, bInit, (flags AND VisuElems.Visu_InputFlags.Password) = 1, 's'); ELSE VisuDlg_CheckedAppend(stOutputValue, stVariableValue, bInit, (flags AND VisuElems.Visu_InputFlags.Password) = 1, 'S'); END_IF, VisuElemId=-1
    hotkey HotkeyInput Id=481114980352, Key=KeyDown=True, KeyName=D, ActionToExecute=Action=STSnippet=IF bShift THEN VisuDlg_CheckedAppend(stOutputValue, stVariableValue, bInit, (flags AND VisuElems.Visu_InputFlags.Password) = 1, 'd'); ELSE VisuDlg_CheckedAppend(stOutputValue, stVariableValue, bInit, (flags AND VisuElems.Visu_InputFlags.Password) = 1, 'D'); END_IF, VisuElemId=-1
    hotkey HotkeyInput Id=481116028928, Key=KeyDown=True, KeyName=F, ActionToExecute=Action=STSnippet=IF bShift THEN VisuDlg_CheckedAppend(stOutputValue, stVariableValue, bInit, (flags AND VisuElems.Visu_InputFlags.Password) = 1, 'f'); ELSE VisuDlg_CheckedAppend(stOutputValue, stVariableValue, bInit, (flags AND VisuElems.Visu_InputFlags.Password) = 1, 'F'); END_IF, VisuElemId=-1
    hotkey HotkeyInput Id=481117077504, Key=KeyDown=True, KeyName=G, ActionToExecute=Action=STSnippet=IF bShift THEN VisuDlg_CheckedAppend(stOutputValue, stVariableValue, bInit, (flags AND VisuElems.Visu_InputFlags.Password) = 1, 'g'); ELSE VisuDlg_CheckedAppend(stOutputValue, stVariableValue, bInit, (flags AND VisuElems.Visu_InputFlags.Password) = 1, 'G'); END_IF, VisuElemId=-1
    hotkey HotkeyInput Id=481118126080, Key=KeyDown=True, KeyName=H, ActionToExecute=Action=STSnippet=IF bShift THEN VisuDlg_CheckedAppend(stOutputValue, stVariableValue, bInit, (flags AND VisuElems.Visu_InputFlags.Password) = 1, 'h'); ELSE VisuDlg_CheckedAppend(stOutputValue, stVariableValue, bInit, (flags AND VisuElems.Visu_InputFlags.Password) = 1, 'H'); END_IF, VisuElemId=-1
    hotkey HotkeyInput Id=481119174656, Key=KeyDown=True, KeyName=J, ActionToExecute=Action=STSnippet=IF bShift THEN VisuDlg_CheckedAppend(stOutputValue, stVariableValue, bInit, (flags AND VisuElems.Visu_InputFlags.Password) = 1, 'j'); ELSE VisuDlg_CheckedAppend(stOutputValue, stVariableValue, bInit, (flags AND VisuElems.Visu_InputFlags.Password) = 1, 'J'); END_IF, VisuElemId=-1
    hotkey HotkeyInput Id=481120223232, Key=KeyDown=True, KeyName=K, ActionToExecute=Action=STSnippet=IF bShift THEN VisuDlg_CheckedAppend(stOutputValue, stVariableValue, bInit, (flags AND VisuElems.Visu_InputFlags.Password) = 1, 'k'); ELSE VisuDlg_CheckedAppend(stOutputValue, stVariableValue, bInit, (flags AND VisuElems.Visu_InputFlags.Password) = 1, 'K'); END_IF, VisuElemId=-1
    hotkey HotkeyInput Id=481121271808, Key=KeyDown=True, KeyName=L, ActionToExecute=Action=STSnippet=IF bShift THEN VisuDlg_CheckedAppend(stOutputValue, stVariableValue, bInit, (flags AND VisuElems.Visu_InputFlags.Password) = 1, 'l'); ELSE VisuDlg_CheckedAppend(stOutputValue, stVariableValue, bInit, (flags AND VisuElems.Visu_InputFlags.Password) = 1, 'L'); END_IF, VisuElemId=-1
    hotkey HotkeyInput Id=481122320384, Key=KeyDown=True, KeyName=Z, ActionToExecute=Action=STSnippet=IF bShift THEN VisuDlg_CheckedAppend(stOutputValue, stVariableValue, bInit, (flags AND VisuElems.Visu_InputFlags.Password) = 1, 'z'); ELSE VisuDlg_CheckedAppend(stOutputValue, stVariableValue, bInit, (flags AND VisuElems.Visu_InputFlags.Password) = 1, 'Z'); END_IF, VisuElemId=-1
    hotkey HotkeyInput Id=481123368960, Key=KeyDown=True, KeyName=X, ActionToExecute=Action=STSnippet=IF bShift THEN VisuDlg_CheckedAppend(stOutputValue, stVariableValue, bInit, (flags AND VisuElems.Visu_InputFlags.Password) = 1, 'x'); ELSE VisuDlg_CheckedAppend(stOutputValue, stVariableValue, bInit, (flags AND VisuElems.Visu_InputFlags.Password) = 1, 'X'); END_IF, VisuElemId=-1
    hotkey HotkeyInput Id=481124417536, Key=KeyDown=True, KeyName=C, ActionToExecute=Action=STSnippet=IF bShift THEN VisuDlg_CheckedAppend(stOutputValue, stVariableValue, bInit, (flags AND VisuElems.Visu_InputFlags.Password) = 1, 'c'); ELSE VisuDlg_CheckedAppend(stOutputValue, stVariableValue, bInit, (flags AND VisuElems.Visu_InputFlags.Password) = 1, 'C'); END_IF, VisuElemId=-1
    hotkey HotkeyInput Id=481125466112, Key=KeyDown=True, KeyName=V, ActionToExecute=Action=STSnippet=IF bShift THEN VisuDlg_CheckedAppend(stOutputValue, stVariableValue, bInit, (flags AND VisuElems.Visu_InputFlags.Password) = 1, 'v'); ELSE VisuDlg_CheckedAppend(stOutputValue, stVariableValue, bInit, (flags AND VisuElems.Visu_InputFlags.Password) = 1, 'V'); END_IF, VisuElemId=-1
    hotkey HotkeyInput Id=481126514688, Key=KeyDown=True, KeyName=B, ActionToExecute=Action=STSnippet=IF bShift THEN VisuDlg_CheckedAppend(stOutputValue, stVariableValue, bInit, (flags AND VisuElems.Visu_InputFlags.Password) = 1, 'b'); ELSE VisuDlg_CheckedAppend(stOutputValue, stVariableValue, bInit, (flags AND VisuElems.Visu_InputFlags.Password) = 1, 'B'); END_IF, VisuElemId=-1
    hotkey HotkeyInput Id=481127563264, Key=KeyDown=True, KeyName=N, ActionToExecute=Action=STSnippet=IF bShift THEN VisuDlg_CheckedAppend(stOutputValue, stVariableValue, bInit, (flags AND VisuElems.Visu_InputFlags.Password) = 1, 'n'); ELSE VisuDlg_CheckedAppend(stOutputValue, stVariableValue, bInit, (flags AND VisuElems.Visu_InputFlags.Password) = 1, 'N'); END_IF, VisuElemId=-1
    hotkey HotkeyInput Id=481128611840, Key=KeyDown=True, KeyName=M, ActionToExecute=Action=STSnippet=IF bShift THEN VisuDlg_CheckedAppend(stOutputValue, stVariableValue, bInit, (flags AND VisuElems.Visu_InputFlags.Password) = 1, 'm'); ELSE VisuDlg_CheckedAppend(stOutputValue, stVariableValue, bInit, (flags AND VisuElems.Visu_InputFlags.Password) = 1, 'M'); END_IF, VisuElemId=-1
    hotkey HotkeyInput Id=481129660416, Key=KeyDown=True, KeyName=COMMA, ActionToExecute=Action=STSnippet=IF bShift THEN VisuDlg_CheckedAppend(stOutputValue, stVariableValue, bInit, (flags AND VisuElems.Visu_InputFlags.Password) = 1, ','); ELSE VisuDlg_CheckedAppend(stOutputValue, stVariableValue, bInit, (flags AND VisuElems.Visu_InputFlags.Password) = 1, '.'); END_IF, VisuElemId=-1
    hotkey HotkeyInput Id=481131757568, Key=KeyDown=True, KeyName=NUM1, ActionToExecute=Action=STSnippet=VisuDlg_CheckedAppend(stOutputValue, stVariableValue, bInit, (flags AND VisuElems.Visu_InputFlags.Password) = 1, '1');, VisuElemId=-1
    hotkey HotkeyInput Id=481132806144, Key=KeyDown=True, KeyName=NUM2, ActionToExecute=Action=STSnippet=VisuDlg_CheckedAppend(stOutputValue, stVariableValue, bInit, (flags AND VisuElems.Visu_InputFlags.Password) = 1, '2');, VisuElemId=-1
    hotkey HotkeyInput Id=481133854720, Key=KeyDown=True, KeyName=NUM3, ActionToExecute=Action=STSnippet=VisuDlg_CheckedAppend(stOutputValue, stVariableValue, bInit, (flags AND VisuElems.Visu_InputFlags.Password) = 1, '3');, VisuElemId=-1
    hotkey HotkeyInput Id=481134903296, Key=KeyDown=True, KeyName=NUM4, ActionToExecute=Action=STSnippet=VisuDlg_CheckedAppend(stOutputValue, stVariableValue, bInit, (flags AND VisuElems.Visu_InputFlags.Password) = 1, '4');, VisuElemId=-1
    hotkey HotkeyInput Id=481135951872, Key=KeyDown=True, KeyName=NUM5, ActionToExecute=Action=STSnippet=VisuDlg_CheckedAppend(stOutputValue, stVariableValue, bInit, (flags AND VisuElems.Visu_InputFlags.Password) = 1, '5');, VisuElemId=-1
    hotkey HotkeyInput Id=481137000448, Key=KeyDown=True, KeyName=NUM6, ActionToExecute=Action=STSnippet=VisuDlg_CheckedAppend(stOutputValue, stVariableValue, bInit, (flags AND VisuElems.Visu_InputFlags.Password) = 1, '6');, VisuElemId=-1
    hotkey HotkeyInput Id=481138049024, Key=KeyDown=True, KeyName=NUM7, ActionToExecute=Action=STSnippet=VisuDlg_CheckedAppend(stOutputValue, stVariableValue, bInit, (flags AND VisuElems.Visu_InputFlags.Password) = 1, '7');, VisuElemId=-1
    hotkey HotkeyInput Id=481139097600, Key=KeyDown=True, KeyName=NUM8, ActionToExecute=Action=STSnippet=VisuDlg_CheckedAppend(stOutputValue, stVariableValue, bInit, (flags AND VisuElems.Visu_InputFlags.Password) = 1, '8');, VisuElemId=-1
    hotkey HotkeyInput Id=481140146176, Key=KeyDown=True, KeyName=NUM9, ActionToExecute=Action=STSnippet=VisuDlg_CheckedAppend(stOutputValue, stVariableValue, bInit, (flags AND VisuElems.Visu_InputFlags.Password) = 1, '9');, VisuElemId=-1
    hotkey HotkeyInput Id=481141194752, Key=KeyDown=True, KeyName=NUM0, ActionToExecute=Action=STSnippet=VisuDlg_CheckedAppend(stOutputValue, stVariableValue, bInit, (flags AND VisuElems.Visu_InputFlags.Password) = 1, '0');, VisuElemId=-1
END_VISUALIZATION

// ---- VISUs/Custom_Numpad.TcVIS
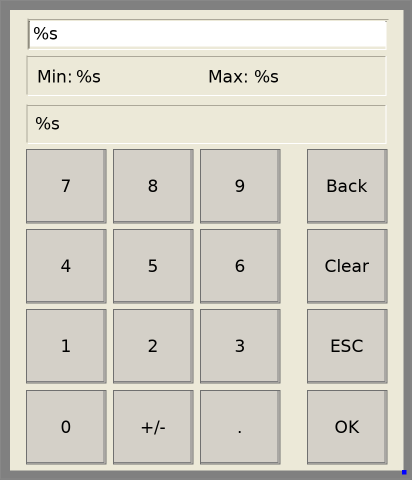
VISUALIZATION Custom_Numpad  // 412x480
VAR_INPUT
	stVariableValue : STRING;
	stMin : STRING;
	stMax : STRING;
	stTitle : STRING;
	flags : DWORD;
END_VAR
VAR
	bInit : BOOL;
	stMessage : STRING;
	stOutputValue : STRING;
END_VAR
    Rectangle (0,0 412x480)
    Rectangle (10,142 393x83)
    Rectangle (10,225 393x80)
    Rectangle (10,305 393x80)
    Rectangle (10,385 393x85)
    Button (307,390 80x74), "OK"
        OnMouseDown: CloseDialog Dialog=Custom_Numpad, Result=OK, NumpadKeypad=True, NumpadKeypadSet=True
    Button (307,309 80x74), "ESC"
        OnMouseDown: CloseDialog Dialog=Custom_Numpad, Result=Cancel, NumpadKeypad=True, NumpadKeypadSet=True
    Button (307,229 80x74), "Clear"
        OnMouseDown: execute {
            stVariableValue := '';
            stOutputValue := '';
            flags := flags AND 16#0008;
            flags := flags AND 16#0010;
        }
    Button (307,149 80x74), "Back"
        OnMouseDown: execute { VisuDlg_CheckedBack(stOutputValue, stVariableValue, bInit); }
    Button (200,390 80x74), "."
        OnMouseDown: execute { VisuDlg_CheckedAppend(stOutputValue, stVariableValue, bInit, (flags AND VisuElems.Visu_InputFlags.Password) = 1, '.'); }
    Button (113,390 80x74), "+/-"
        OnMouseDown: execute { VisuDlg_CheckedChangeSign(stOutputValue, stVariableValue, bInit, (flags AND VisuElems.Visu_InputFlags.Password) = 1); }
    Button (26,390 80x74), "0"
        OnMouseDown: execute { VisuDlg_CheckedAppend(stOutputValue, stVariableValue, bInit, (flags AND VisuElems.Visu_InputFlags.Password) = 1, '0'); }
    Button (26,309 80x74), "1"
        OnMouseDown: execute { VisuDlg_CheckedAppend(stOutputValue, stVariableValue, bInit, (flags AND VisuElems.Visu_InputFlags.Password) = 1, '1'); }
    Button (113,309 80x74), "2"
        OnMouseDown: execute { VisuDlg_CheckedAppend(stOutputValue, stVariableValue, bInit, (flags AND VisuElems.Visu_InputFlags.Password) = 1, '2'); }
    Button (200,309 80x74), "3"
        OnMouseDown: execute { VisuDlg_CheckedAppend(stOutputValue, stVariableValue, bInit, (flags AND VisuElems.Visu_InputFlags.Password) = 1, '3'); }
    Button (26,229 80x74), "4"
        OnMouseDown: execute { VisuDlg_CheckedAppend(stOutputValue, stVariableValue, bInit, (flags AND VisuElems.Visu_InputFlags.Password) = 1, '4'); }
    Button (113,229 80x74), "5"
        OnMouseDown: execute { VisuDlg_CheckedAppend(stOutputValue, stVariableValue, bInit, (flags AND VisuElems.Visu_InputFlags.Password) = 1, '5'); }
    Button (200,229 80x74), "6"
        OnMouseDown: execute { VisuDlg_CheckedAppend(stOutputValue, stVariableValue, bInit, (flags AND VisuElems.Visu_InputFlags.Password) = 1, '6'); }
    Button (26,149 80x74), "7"
        OnMouseDown: execute { VisuDlg_CheckedAppend(stOutputValue, stVariableValue, bInit, (flags AND VisuElems.Visu_InputFlags.Password) = 1, '7'); }
    Button (113,149 80x74), "8"
        OnMouseDown: execute { VisuDlg_CheckedAppend(stOutputValue, stVariableValue, bInit, (flags AND VisuElems.Visu_InputFlags.Password) = 1, '8'); }
    Button (200,149 80x74), "9"
        OnMouseDown: execute { VisuDlg_CheckedAppend(stOutputValue, stVariableValue, bInit, (flags AND VisuElems.Visu_InputFlags.Password) = 1, '9'); }
    Rectangle (10,10 393x48)
    Rectangle (10,57 393x85)
    Rectangle (73,64 127x25), "%s", text variable: stMin, invisible if: LEN(stMin) = 0
    Rectangle (251,64 127x25), "%s", text variable: stMax, invisible if: LEN(stMax) = 0
    Rectangle (205,64 45x25), "Max:", text variable: stMin, invisible if: LEN(stMax) = 0
        p55702900: SEL(((UDINT_TO_DINT(flags AND 16#0010))=16#0010),16#FF000000,16#FFFF0000)
    Rectangle (402,470 4x4)
    Polyline (27,94) (27,56) (385,56)
    Polyline (27,142) (27,105) (385,105)
    Polyline (28,49) (28,19) (388,19)
    Polyline (28,143) (386,143) (386,105)
    Polyline (28,95) (386,95) (386,56)
    Polyline (29,49) (386,49) (386,21)
    Polyline (29,48) (29,21) (386,21)
    Rectangle (32,111 349x25), "%s", text variable: stMessage
    Rectangle (34,64 41x25), "Min:", text variable: stMin, invisible if: LEN(stMin) = 0
        p55702900: SEL(((UDINT_TO_DINT(flags AND 16#0008))=16#0008),16#FF000000,16#FFFF0000)
    Rectangle (30,21 355x25), "%s", text variable: stOutputValue
    hotkey HotkeyInput Id=481049968640, Key=KeyDown=True, KeyName=0, ActionToExecute=Action=STSnippet=VisuDlg_CheckedAppend(stOutputValue, stVariableValue, bInit, (flags AND VisuElems.Visu_InputFlags.Password) = 1, '0');, VisuElemId=-1
    hotkey HotkeyInput Id=481053114368, Key=KeyDown=True, KeyName=NUM0, ActionToExecute=Action=STSnippet=VisuDlg_CheckedAppend(stOutputValue, stVariableValue, bInit, (flags AND VisuElems.Visu_InputFlags.Password) = 1, '0');, VisuElemId=-1
    hotkey HotkeyInput Id=481054162944, Key=KeyDown=True, KeyName=1, ActionToExecute=Action=STSnippet=VisuDlg_CheckedAppend(stOutputValue, stVariableValue, bInit, (flags AND VisuElems.Visu_InputFlags.Password) = 1, '1');, VisuElemId=-1
    hotkey HotkeyInput Id=481055211520, Key=KeyDown=True, KeyName=NUM1, ActionToExecute=Action=STSnippet=VisuDlg_CheckedAppend(stOutputValue, stVariableValue, bInit, (flags AND VisuElems.Visu_InputFlags.Password) = 1, '1');, VisuElemId=-1
    hotkey HotkeyInput Id=481056260096, Key=KeyDown=True, KeyName=2, ActionToExecute=Action=STSnippet=VisuDlg_CheckedAppend(stOutputValue, stVariableValue, bInit, (flags AND VisuElems.Visu_InputFlags.Password) = 1, '2');, VisuElemId=-1
    hotkey HotkeyInput Id=481057308672, Key=KeyDown=True, KeyName=NUM2, ActionToExecute=Action=STSnippet=VisuDlg_CheckedAppend(stOutputValue, stVariableValue, bInit, (flags AND VisuElems.Visu_InputFlags.Password) = 1, '2');, VisuElemId=-1
    hotkey HotkeyInput Id=481058357248, Key=KeyDown=True, KeyName=3, ActionToExecute=Action=STSnippet=VisuDlg_CheckedAppend(stOutputValue, stVariableValue, bInit, (flags AND VisuElems.Visu_InputFlags.Password) = 1, '3');, VisuElemId=-1
    hotkey HotkeyInput Id=481059405824, Key=KeyDown=True, KeyName=NUM3, ActionToExecute=Action=STSnippet=VisuDlg_CheckedAppend(stOutputValue, stVariableValue, bInit, (flags AND VisuElems.Visu_InputFlags.Password) = 1, '3');, VisuElemId=-1
    hotkey HotkeyInput Id=481060454400, Key=KeyDown=True, KeyName=4, ActionToExecute=Action=STSnippet=VisuDlg_CheckedAppend(stOutputValue, stVariableValue, bInit, (flags AND VisuElems.Visu_InputFlags.Password) = 1, '4');, VisuElemId=-1
    hotkey HotkeyInput Id=481061502976, Key=KeyDown=True, KeyName=NUM4, ActionToExecute=Action=STSnippet=VisuDlg_CheckedAppend(stOutputValue, stVariableValue, bInit, (flags AND VisuElems.Visu_InputFlags.Password) = 1, '4');, VisuElemId=-1
    hotkey HotkeyInput Id=481062551552, Key=KeyDown=True, KeyName=5, ActionToExecute=Action=STSnippet=VisuDlg_CheckedAppend(stOutputValue, stVariableValue, bInit, (flags AND VisuElems.Visu_InputFlags.Password) = 1, '5');, VisuElemId=-1
    hotkey HotkeyInput Id=481063600128, Key=KeyDown=True, KeyName=NUM5, ActionToExecute=Action=STSnippet=VisuDlg_CheckedAppend(stOutputValue, stVariableValue, bInit, (flags AND VisuElems.Visu_InputFlags.Password) = 1, '5');, VisuElemId=-1
    hotkey HotkeyInput Id=481064648704, Key=KeyDown=True, KeyName=6, ActionToExecute=Action=STSnippet=VisuDlg_CheckedAppend(stOutputValue, stVariableValue, bInit, (flags AND VisuElems.Visu_InputFlags.Password) = 1, '6');, VisuElemId=-1
    hotkey HotkeyInput Id=481065697280, Key=KeyDown=True, KeyName=NUM6, ActionToExecute=Action=STSnippet=VisuDlg_CheckedAppend(stOutputValue, stVariableValue, bInit, (flags AND VisuElems.Visu_InputFlags.Password) = 1, '6');, VisuElemId=-1
    hotkey HotkeyInput Id=481066745856, Key=KeyDown=True, KeyName=7, ActionToExecute=Action=STSnippet=VisuDlg_CheckedAppend(stOutputValue, stVariableValue, bInit, (flags AND VisuElems.Visu_InputFlags.Password) = 1, '7');, VisuElemId=-1
    hotkey HotkeyInput Id=481067794432, Key=KeyDown=True, KeyName=NUM7, ActionToExecute=Action=STSnippet=VisuDlg_CheckedAppend(stOutputValue, stVariableValue, bInit, (flags AND VisuElems.Visu_InputFlags.Password) = 1, '7');, VisuElemId=-1
    hotkey HotkeyInput Id=481068843008, Key=KeyDown=True, KeyName=8, ActionToExecute=Action=STSnippet=VisuDlg_CheckedAppend(stOutputValue, stVariableValue, bInit, (flags AND VisuElems.Visu_InputFlags.Password) = 1, '8');, VisuElemId=-1
    hotkey HotkeyInput Id=481069891584, Key=KeyDown=True, KeyName=NUM8, ActionToExecute=Action=STSnippet=VisuDlg_CheckedAppend(stOutputValue, stVariableValue, bInit, (flags AND VisuElems.Visu_InputFlags.Password) = 1, '8');, VisuElemId=-1
    hotkey HotkeyInput Id=481070940160, Key=KeyDown=True, KeyName=9, ActionToExecute=Action=STSnippet=VisuDlg_CheckedAppend(stOutputValue, stVariableValue, bInit, (flags AND VisuElems.Visu_InputFlags.Password) = 1, '9');, VisuElemId=-1
    hotkey HotkeyInput Id=481071988736, Key=KeyDown=True, KeyName=NUM9, ActionToExecute=Action=STSnippet=VisuDlg_CheckedAppend(stOutputValue, stVariableValue, bInit, (flags AND VisuElems.Visu_InputFlags.Password) = 1, '9');, VisuElemId=-1
    hotkey HotkeyInput Id=481073037312, Key=KeyDown=True, KeyName=SUBTRACT, ActionToExecute=Action=STSnippet=VisuDlg_CheckedChangeSign(stOutputValue, stVariableValue, bInit, (flags AND VisuElems.Visu_InputFlags.Password) = 1);, VisuElemId=-1
    hotkey HotkeyInput Id=481074085888, Key=KeyDown=True, KeyName=COMMA, ActionToExecute=Action=STSnippet=VisuDlg_CheckedAppend(stOutputValue, stVariableValue, bInit, (flags AND VisuElems.Visu_InputFlags.Password) = 1, '.');, VisuElemId=-1
    hotkey HotkeyInput Id=481075134464, Key=KeyDown=True, KeyName=BACKSPACE, ActionToExecute=Action=STSnippet=VisuDlg_CheckedBack(stOutputValue, stVariableValue, bInit);, VisuElemId=-1
    hotkey HotkeyInput Id=481076183040, Key=KeyDown=True, KeyName=DELETE, ActionToExecute=Action=STSnippet=stVariableValue := ''; stOutputValue := ''; flags := flags AND 16#0008; flags := flags AND 16#0010;, VisuElemId=-1
    hotkey HotkeyInput Id=481077231616, Key=KeyDown=True, KeyName=ESCAPE, ActionToExecute=Action=Dialog=Custom_Numpad, Result=Cancel, NumpadKeypad=True, NumpadKeypadSet=True, VisuElemId=-1
    hotkey HotkeyInput Id=481078280192, Key=KeyDown=True, KeyName=RETURN_KEY, ActionToExecute=Action=Dialog=Custom_Numpad, Result=OK, NumpadKeypad=True, NumpadKeypadSet=True, VisuElemId=-1
END_VISUALIZATION

// ---- VISUs/Visualization.TcVIS
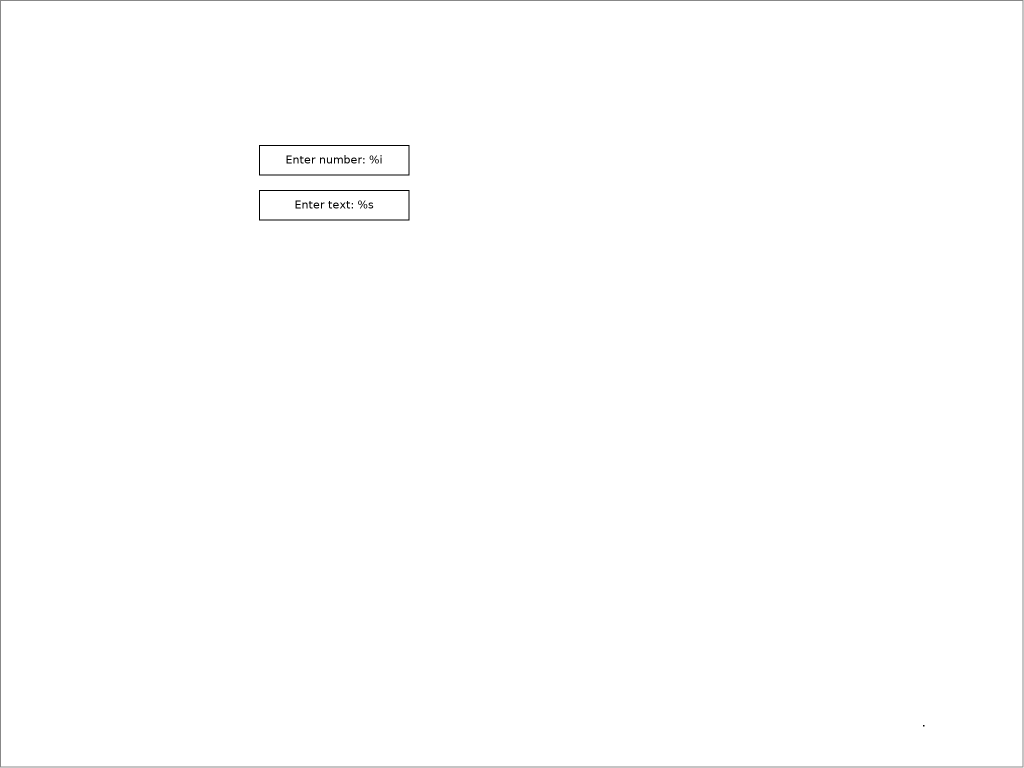
VISUALIZATION Visualization  // 1024x768
    Rectangle (259,145 150x30), "Enter number: %i", text variable: MAIN.iTest
        OnMouseDown: write the text variable via Default
    Rectangle (259,190 150x30), "Enter text: %s", text variable: MAIN.sTest
        OnMouseDown: write the text variable via Default
    Rectangle (923,725 1x1)
END_VISUALIZATION
